FUNCTION_BLOCK DrawAxis EXTENDS FB_PackML_BaseModule
VAR
	Axis	   : FB_Component_BasicSlaveAxis := (Name := 'Unwind');
	_MasterRef : REFERENCE TO AXIS_REF;
END_VAR

METHOD PROTECTED Aborting
//Mode is ignored
CASE SequenceState OF
	0:
		NoStateTasksToComplete := FALSE;

		// Stop Axis
		Axis.Override := 100;
		IF Axis.Stop() OR Axis.Error THEN //This will also GearOut
			SequenceState := SequenceState + 10;
		END_IF

	10:
		IF Axis.Stopped THEN
			SequenceState := SequenceState + 10;
		END_IF

	20: // Disable Axis
		IF Axis.Disable() THEN
			SequenceState := SequenceState + 10;
		END_IF

	30:
		IF NOT Axis.Enabled THEN
			SequenceState := SequenceState + 10;
		END_IF

	40:
		StateTasksComplete := TRUE;
END_CASE

SUPER^.Aborting();
END_METHOD

PROPERTY AxisRef : REFERENCE TO AXIS_REF
GET
AxisRef REF= Axis.Axis;
END_GET
END_PROPERTY

METHOD PROTECTED Completing
VAR_INST
	StopAxis : BOOL;
END_VAR
CASE _CurrentMode OF
	ePMLUnitMode_Production:
		CASE SequenceState OF
			0:
				NoStateTasksToComplete := FALSE;
				IF Axis.InGear AND_THEN Axis.Master1.Status.StandStill THEN //Wait for Master Axis to Stop
					StopAxis := TRUE;
				ELSIF NOT Axis.InGear THEN
					StopAxis := TRUE;
				ELSE
					StopAxis := FALSE;
				END_IF

				IF StopAxis AND_THEN Axis.Stop() THEN // This will also GearOut
					SequenceState := SequenceState + 10;
				END_IF

			10:
				IF Axis.Stopped THEN
					SequenceState := SequenceState + 10;
				END_IF

			20:
				StateTasksComplete := TRUE;
		END_CASE

	ePMLProtUnitMode_Maintenance, ePMLProtUnitMode_Manual:
		;
END_CASE

SUPER^.Completing();
END_METHOD

METHOD PUBLIC CyclicLogic
IF NOT InitComplete THEN
	_InitComplete := Initialize();
	RETURN;
END_IF

SUPER^.CyclicLogic();
END_METHOD

METHOD PROTECTED Initialize : BOOL;
Initialize := FALSE;
CASE DescendantSequenceState OF
	0:
		RegisterComponent(Axis);
		DescendantSequenceState := DescendantSequenceState + 10;

	10:
		IF SUPER^.Initialize() THEN
			DescendantSequenceState := DescendantSequenceState + 10;
		END_IF

	20:
		Initialize := TRUE;
END_CASE
END_METHOD

PROPERTY MasterAxisRef : REFERENCE TO AXIS_REF
SET
_MasterRef REF= MasterAxisRef;
END_SET
END_PROPERTY

METHOD PROTECTED Starting
CASE _CommandedMode OF
	ePMLProtUnitMode_Production:
		CASE SequenceState OF
			0:
				NoStateTasksToComplete := FALSE;
				IF Axis.Enable() THEN
					SequenceState := SequenceState + 10;
				END_IF

			10:
				IF Axis.Enabled THEN
					SequenceState := SequenceState + 10;
				END_IF

			20:
				Axis.Master1 REF= _MasterRef;
				IF Axis.GearIn() THEN
					SequenceState := SequenceState + 10;
				END_IF

			30:
				IF Axis.InGear THEN
					SequenceState := SequenceState + 10;
				END_IF

			40:
				StateTasksComplete := TRUE;
		END_CASE
END_CASE

SUPER^.Starting();
END_METHOD

METHOD PROTECTED Stopping
CASE _CurrentMode OF
	ePMLUnitMode_Production:
		CASE SequenceState OF
			0:
				NoStateTasksToComplete := FALSE;
				IF Axis.Stop() THEN //This will also GearOut
					SequenceState := SequenceState + 10;
				END_IF

			10:
				IF Axis.Stopped THEN
					SequenceState := SequenceState + 10;
				END_IF

			20:
				StateTasksComplete := TRUE;
		END_CASE
END_CASE

SUPER^.Stopping();
END_METHOD

END_FUNCTION_BLOCK

(* stored: Version 1.1.0.1, ProductVersion 3.1.4024.12
   POU DrawAxis: Id {6f7f3fdd-1761-46b2-a834-6c3784a9206a}, SpecialFunc None
   Folder Acting States: Id {ac03b756-ae75-4ddc-8701-cd226ef523c7}
   Folder CyclicLogic: Id {20c2e56f-0469-4216-ab80-31915d3aec52}
   Folder Initialize: Id {4ca6b6de-8013-4e81-9476-05982f2562f6}
   Method Aborting: Id {d947f5e2-2d16-49a5-9815-3f039233a9f0}
   Property AxisRef: Id {6a546205-aa1a-4058-a964-b861546a6b3a}
   Get Get: Id {c2ba8eac-8f12-4d77-bfd7-5fb7b5eee94d}
   Method Completing: Id {1a88739c-e241-40e6-932c-4e770d465d42}
   Method CyclicLogic: Id {071f67bd-24e9-4734-8fa9-d70acebb508f}
   Method Initialize: Id {aa1d8f3c-de5d-440d-88b2-cf20a1bca6eb}
   Property MasterAxisRef: Id {c8aeeb47-6497-45ee-b23a-b03bca698c96}
   Set Set: Id {4c5a7eeb-c2c9-4a9d-9b74-c57a2ad6979d}
   Method Starting: Id {08b85550-4819-4b11-b046-f4ec48d539b6}
   Method Stopping: Id {2444f023-ed59-4632-8f42-8076dedaa106} *)
